FUNCTION_BLOCK ABSTRACT tempSensor
VAR
	rawValue			AT %I*	: INT;		// resistance measurement value of sensor
END_VAR
(*~
<docu>
	<summary>
			Abstract implementation of a Temperature sensor class
			Usage as follows :
			<code>
				FUNCTION_BLOCK concreteTempSensor EXTENDS tempSensor
			</code>
	</summary>				
</docu>	
~*)

END_FUNCTION_BLOCK

(* stored: Version 1.1.0.1, ProductVersion 3.1.4024.12
   POU FB_TempSensor: Id {d20820a4-0d8a-43f0-b4e4-a3d10b2764cf}, SpecialFunc None *)
